// TIA Portal V15.1 export
// export: Created 2020-06-12T07:35:55.1474609Z, ExportSetting None, DisplayName Totally Integrated Automation Portal, DisplayVersion V15.1, DisplayName TIA Portal Openness, DisplayVersion V15.1, DisplayName STEP 7 Professional, DisplayVersion V15.1, DisplayName STEP 7 Safety, DisplayVersion V15.1, DisplayName WinCC Advanced, DisplayVersion V15.1
FUNCTION "Desk_ES1GT07" : Void   // FC166, FBD
{ S7_Optimized_Access := 'TRUE' }
// stored: SetENOAutomatically False
BEGIN

REGION Network 1: ES1GT07 IPB: Desk is on
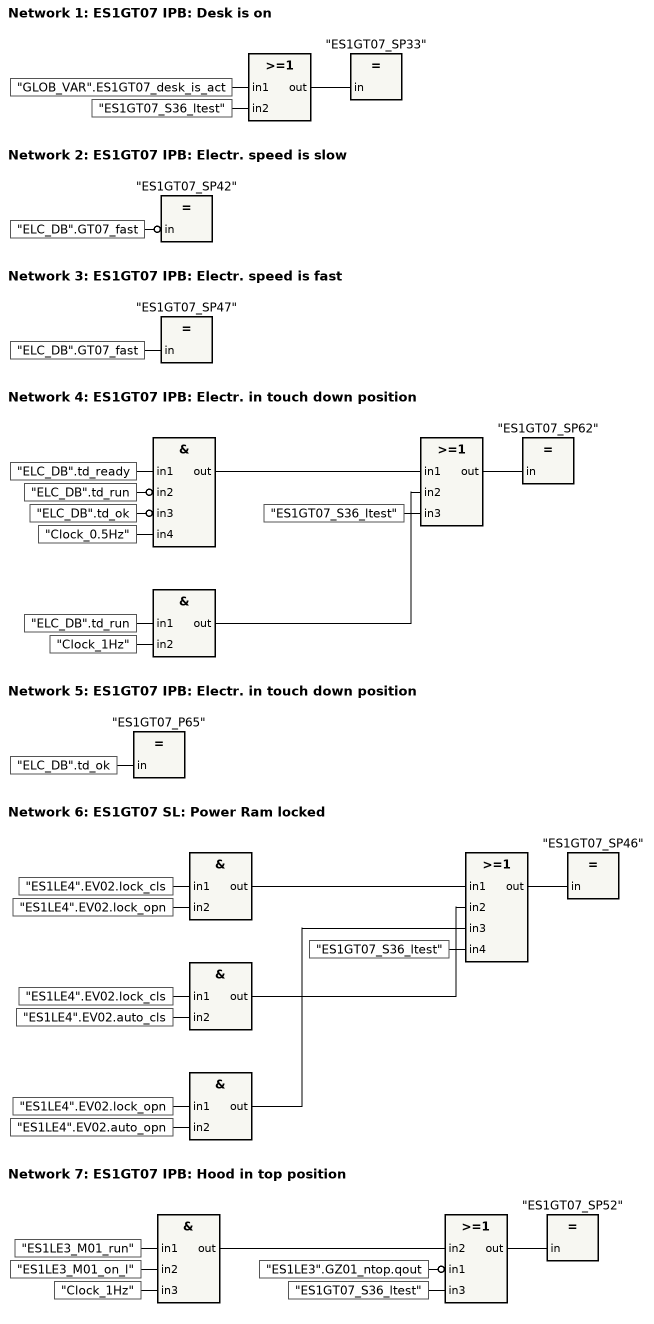
   "ES1GT07_SP33" := "GLOB_VAR".ES1GT07_desk_is_act OR "ES1GT07_S36_ltest";
END_REGION

REGION Network 2: ES1GT07 IPB: Electr. speed is slow
   "ES1GT07_SP42" := NOT "ELC_DB".GT07_fast;
END_REGION

REGION Network 3: ES1GT07 IPB: Electr. speed is fast
   "ES1GT07_SP47" := "ELC_DB".GT07_fast;
END_REGION

REGION Network 4: ES1GT07 IPB: Electr. in touch down position
   "ES1GT07_SP62" := ("ELC_DB".td_ready AND NOT "ELC_DB".td_run AND NOT "ELC_DB".td_ok AND "Clock_0.5Hz") OR ("ELC_DB".td_run AND "Clock_1Hz") OR "ES1GT07_S36_ltest";
END_REGION

REGION Network 5: ES1GT07 IPB: Electr. in touch down position
   "ES1GT07_P65" := "ELC_DB".td_ok;
END_REGION

REGION Network 6: ES1GT07 SL: Power Ram locked
   "ES1GT07_SP46" := ("ES1LE4".EV02.lock_cls AND "ES1LE4".EV02.lock_opn) OR ("ES1LE4".EV02.lock_cls AND "ES1LE4".EV02.auto_cls) OR ("ES1LE4".EV02.lock_opn AND "ES1LE4".EV02.auto_opn) OR "ES1GT07_S36_ltest";
END_REGION

REGION Network 7: ES1GT07 IPB: Hood in top position
   "ES1GT07_SP52" := ("ES1LE3_M01_run" AND "ES1LE3_M01_on_l" AND "Clock_1Hz") OR NOT "ES1LE3".GZ01_ntop.qout OR "ES1GT07_S36_ltest";
END_REGION

REGION Network 8: ES1GT07 IPB: Hood in bottom position
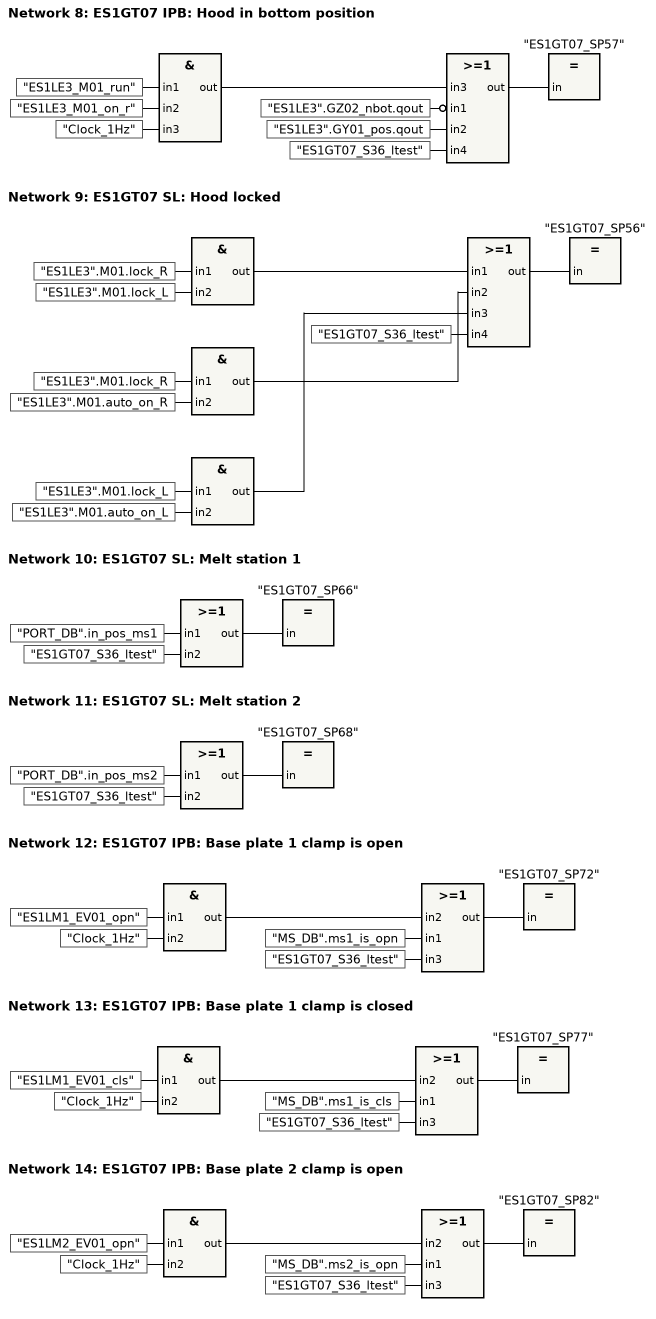
   "ES1GT07_SP57" := ("ES1LE3_M01_run" AND "ES1LE3_M01_on_r" AND "Clock_1Hz") OR NOT "ES1LE3".GZ02_nbot.qout OR "ES1LE3".GY01_pos.qout OR "ES1GT07_S36_ltest";
END_REGION

REGION Network 9: ES1GT07 SL: Hood locked
   // Eh????
   "ES1GT07_SP56" := ("ES1LE3".M01.lock_R AND "ES1LE3".M01.lock_L) OR ("ES1LE3".M01.lock_R AND "ES1LE3".M01.auto_on_R) OR ("ES1LE3".M01.lock_L AND "ES1LE3".M01.auto_on_L) OR "ES1GT07_S36_ltest";
END_REGION

REGION Network 10: ES1GT07 SL: Melt station 1
   "ES1GT07_SP66" := "PORT_DB".in_pos_ms1 OR "ES1GT07_S36_ltest";
END_REGION

REGION Network 11: ES1GT07 SL: Melt station 2
   "ES1GT07_SP68" := "PORT_DB".in_pos_ms2 OR "ES1GT07_S36_ltest";
END_REGION

REGION Network 12: ES1GT07 IPB: Base plate 1 clamp is open
   "ES1GT07_SP72" := ("ES1LM1_EV01_opn" AND "Clock_1Hz") OR "MS_DB".ms1_is_opn OR "ES1GT07_S36_ltest";
END_REGION

REGION Network 13: ES1GT07 IPB: Base plate 1 clamp is closed
   "ES1GT07_SP77" := ("ES1LM1_EV01_cls" AND "Clock_1Hz") OR "MS_DB".ms1_is_cls OR "ES1GT07_S36_ltest";
END_REGION

REGION Network 14: ES1GT07 IPB: Base plate 2 clamp is open
   "ES1GT07_SP82" := ("ES1LM2_EV01_opn" AND "Clock_1Hz") OR "MS_DB".ms2_is_opn OR "ES1GT07_S36_ltest";
END_REGION

REGION Network 15: ES1GT07 IPB: Base plate 2 clamp is closed
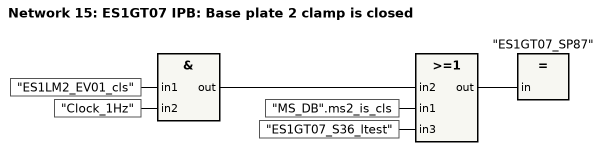
   "ES1GT07_SP87" := ("ES1LM2_EV01_cls" AND "Clock_1Hz") OR "MS_DB".ms2_is_cls OR "ES1GT07_S36_ltest";
END_REGION
END_FUNCTION
